TYPE ST_AutoProvisioning :
	STRUCT
		sType	: STRING;
		sRealm	: STRING;
		sError	: STRING;
	END_STRUCT
END_TYPE

(* stored: Version 1.1.0.1, ProductVersion 3.1.4026.18
   DUT ST_AutoProvisioning: Id {a73040ef-81ec-4b3b-94af-168bb18347a1} *)
